(* PLC project Lib2dMath, Beckhoff Automation GmbH TwinCAT PLC Control 3.5.13.21 *)
(* stored: creationDateTime 2024-03-30T11:42:10.9132946, modificationDateTime 2024-03-30T11:42:10.9579594 *)

FUNCTION fbCalcWinkelvVector : LReal
VAR_INPUT
	Vec:udtVector;
END_VAR
VAR_OUTPUT
	Len:LREAL;
END_VAR
VAR
	ZwErg: LREAL;
END_VAR

            IF ABS(Vec.v.x) > ABS(Vec.v.y) THEN
   ZwErg :=SEL(Vec.v.x<0.0,ATAN(Vec.v.y/vec.v.x),ATAN(Vec.v.y/vec.v.x)+pi);
   len:=Vec.v.x/COS(ZwErg);
   fbCalcWinkelvVector := ZwErg+pi*2.0-DINT_TO_REAL(TRUNC(Zwerg/pi*0.5+1.5))*pi*2.0;
ELSIF ABS(Vec.v.y) > epsilon THEN
    fbCalcWinkelvVector := SEL(Vec.v.y < 0.0,ATAN(-Vec.v.x/vec.v.y)+0.5*pi,ATAN(-Vec.v.x/vec.v.y)-0.5*pi);
   len:=Vec.v.y/SIN(fbCalcWinkelvVector);
else
   fbCalcWinkelvVector :=0.0;
   Len := 0.0;
end_if;
          
END_FUNCTION
